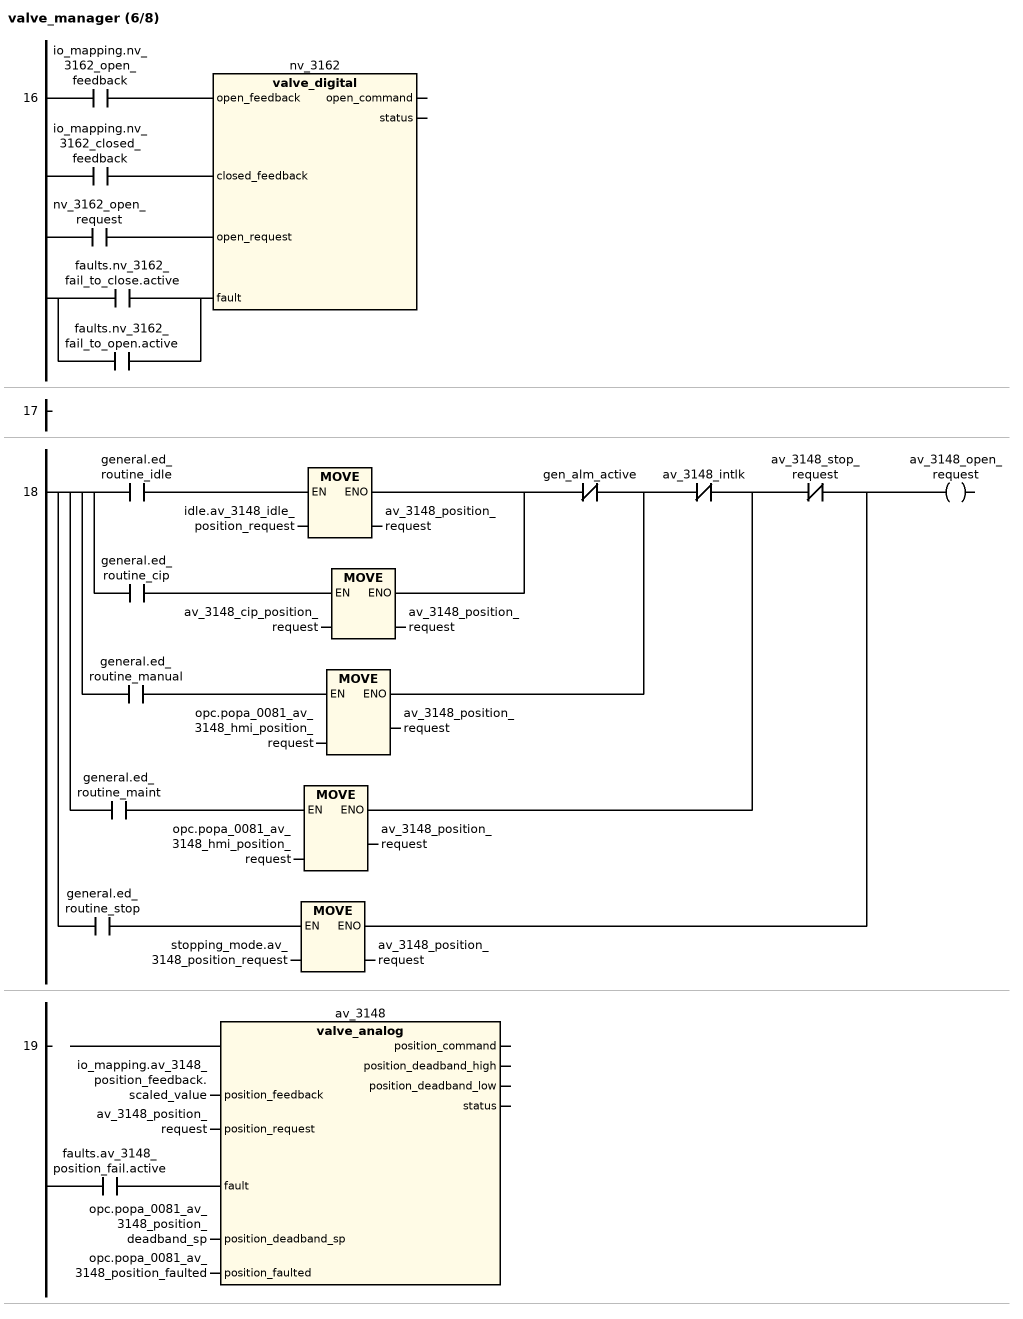
// NETWORK 16
nv_3162(
    open_feedback := io_mapping.nv_3162_open_feedback,
    closed_feedback := io_mapping.nv_3162_closed_feedback,
    open_request := nv_3162_open_request,
    fault := faults.nv_3162_fail_to_close.active OR faults.nv_3162_fail_to_open.active); // valve_digital

// NETWORK 17

// NETWORK 18
_w1 := general.ed_routine_idle;
IF _w1 THEN av_3148_position_request := idle.av_3148_idle_position_request; END_IF
_w2 := general.ed_routine_cip;
IF _w2 THEN av_3148_position_request := av_3148_cip_position_request; END_IF
_w3 := general.ed_routine_manual;
IF _w3 THEN av_3148_position_request := opc.popa_0081_av_3148_hmi_position_request; END_IF
_w4 := general.ed_routine_maint;
IF _w4 THEN av_3148_position_request := opc.popa_0081_av_3148_hmi_position_request; END_IF
_w5 := general.ed_routine_stop;
IF _w5 THEN av_3148_position_request := stopping_mode.av_3148_position_request; END_IF
av_3148_open_request := (((_w1 OR _w2) AND NOT gen_alm_active OR _w3) AND NOT av_3148_intlk OR _w4) AND NOT av_3148_stop_request OR _w5;

// NETWORK 19
av_3148(
    position_feedback := io_mapping.av_3148_position_feedback.scaled_value,
    position_request := av_3148_position_request,
    fault := faults.av_3148_position_fail.active,
    position_deadband_sp := opc.popa_0081_av_3148_position_deadband_sp,
    position_faulted := opc.popa_0081_av_3148_position_faulted); // valve_analog

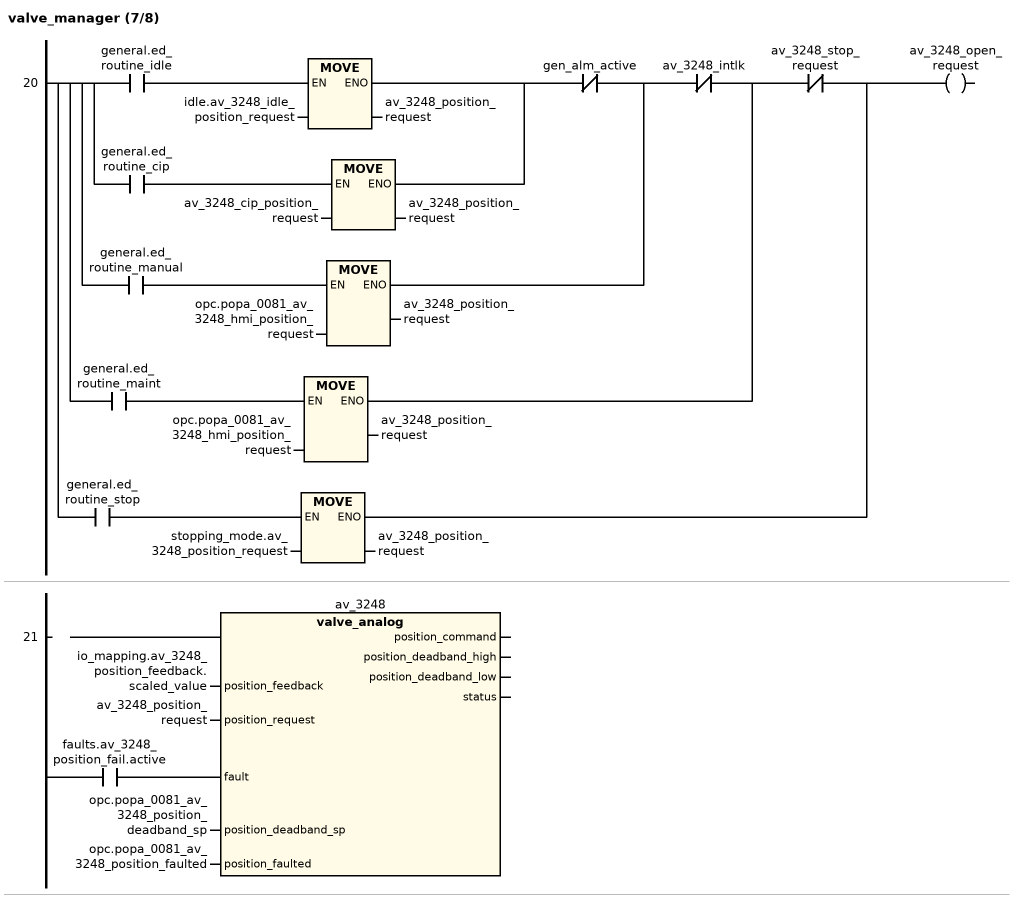
// NETWORK 20
_w6 := general.ed_routine_idle;
IF _w6 THEN av_3248_position_request := idle.av_3248_idle_position_request; END_IF
_w7 := general.ed_routine_cip;
IF _w7 THEN av_3248_position_request := av_3248_cip_position_request; END_IF
_w8 := general.ed_routine_manual;
IF _w8 THEN av_3248_position_request := opc.popa_0081_av_3248_hmi_position_request; END_IF
_w9 := general.ed_routine_maint;
IF _w9 THEN av_3248_position_request := opc.popa_0081_av_3248_hmi_position_request; END_IF
_w10 := general.ed_routine_stop;
IF _w10 THEN av_3248_position_request := stopping_mode.av_3248_position_request; END_IF
av_3248_open_request := (((_w6 OR _w7) AND NOT gen_alm_active OR _w8) AND NOT av_3248_intlk OR _w9) AND NOT av_3248_stop_request OR _w10;

// NETWORK 21
av_3248(
    position_feedback := io_mapping.av_3248_position_feedback.scaled_value,
    position_request := av_3248_position_request,
    fault := faults.av_3248_position_fail.active,
    position_deadband_sp := opc.popa_0081_av_3248_position_deadband_sp,
    position_faulted := opc.popa_0081_av_3248_position_faulted); // valve_analog

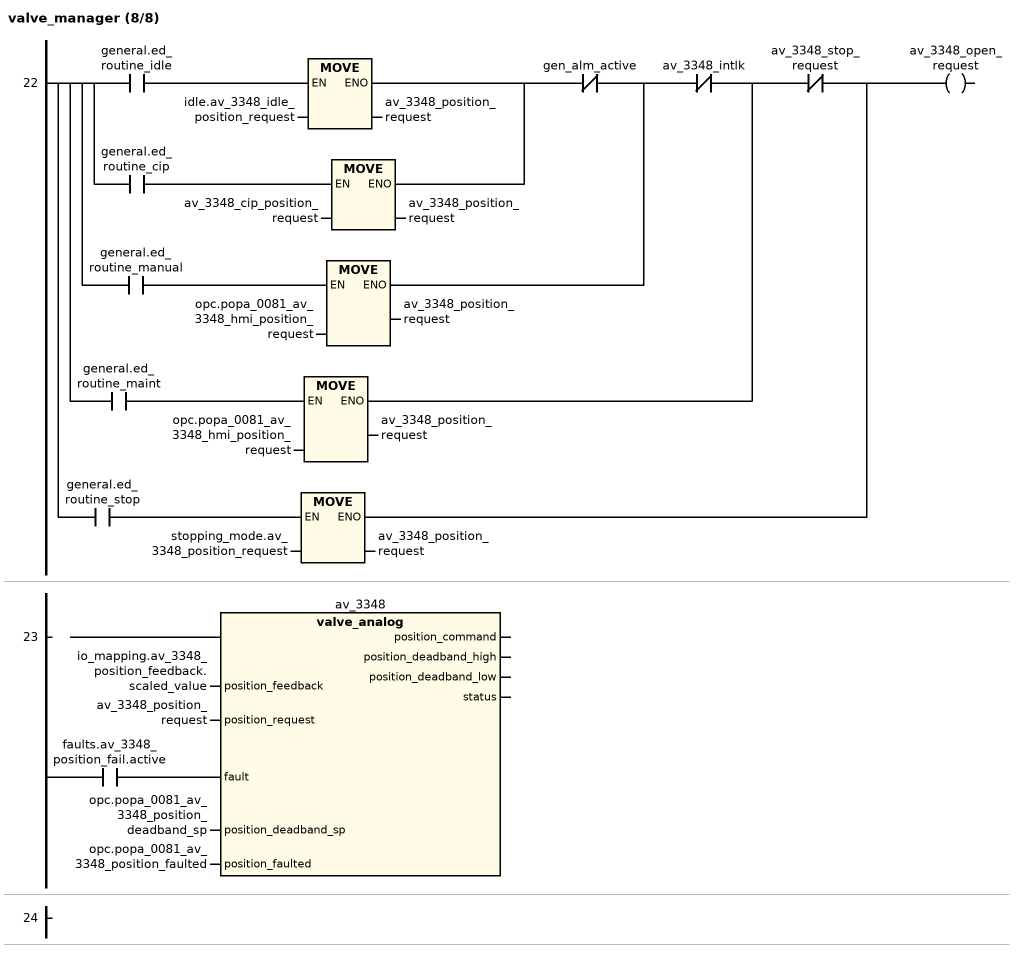
// NETWORK 22
_w11 := general.ed_routine_idle;
IF _w11 THEN av_3348_position_request := idle.av_3348_idle_position_request; END_IF
_w12 := general.ed_routine_cip;
IF _w12 THEN av_3348_position_request := av_3348_cip_position_request; END_IF
_w13 := general.ed_routine_manual;
IF _w13 THEN av_3348_position_request := opc.popa_0081_av_3348_hmi_position_request; END_IF
_w14 := general.ed_routine_maint;
IF _w14 THEN av_3348_position_request := opc.popa_0081_av_3348_hmi_position_request; END_IF
_w15 := general.ed_routine_stop;
IF _w15 THEN av_3348_position_request := stopping_mode.av_3348_position_request; END_IF
av_3348_open_request := (((_w11 OR _w12) AND NOT gen_alm_active OR _w13) AND NOT av_3348_intlk OR _w14) AND NOT av_3348_stop_request OR _w15;

// NETWORK 23
av_3348(
    position_feedback := io_mapping.av_3348_position_feedback.scaled_value,
    position_request := av_3348_position_request,
    fault := faults.av_3348_position_fail.active,
    position_deadband_sp := opc.popa_0081_av_3348_position_deadband_sp,
    position_faulted := opc.popa_0081_av_3348_position_faulted); // valve_analog

// NETWORK 24

END_PROGRAM

// ---- POUs/opc_mapping.TcPOU
PROGRAM opc_mapping
VAR
END_VAR

//This program maps values from the local variable to the OPC readable tag.
//Setpoints should NOT be mapped here.  The OPC tag should be used directly where needed
opc.popa_0081_av_3148_position_fail_active :=faults.av_3148_position_fail.active;
opc.popa_0081_u_3112_fail_to_start_active:=faults.u_3112_fail_to_start.active;
opc.popa_0081_u_3112_fail_to_stop_active:=faults.u_3112_fail_to_stop.active;
opc.popa_0081_u_3160_fail_to_start_active:=faults.u_3160_fail_to_start.active;
opc.popa_0081_u_3160_fail_to_stop_active:=faults.u_3112_fail_to_stop.active;
opc.popa_0081_cpt_3144_low_low_active:=faults.cpt_3144_low_low.active;
opc.popa_0081_cpt_3144_low_active:=faults.cpt_3144_low.active;
opc.popa_0081_cpt_3144_high_active:=faults.cpt_3144_high.active;
opc.popa_0081_cpt_3144_high_high_active:=faults.cpt_3144_high_high.active;

opc.popa_0081_ed_routine_critical_stop := general.ed_critical_stop;
opc.popa_0081_ed_routine_stop := general.ed_routine_stop;
opc.popa_0081_ed_routine_idle := general.ed_routine_idle;
opc.popa_0081_ed_routine_maint := general.ed_routine_maint;
opc.popa_0081_ed_routine_cip := general.ed_routine_cip;

opc.popa_0081_system_date_time_year:=general.system_date_time.year;
opc.popa_0081_system_date_time_month:=general.system_date_time.month;
opc.popa_0081_system_date_time_day:=general.system_date_time.day;
opc.popa_0081_system_date_time_hour:=general.system_date_time.hour;
opc.popa_0081_system_date_time_minute:=general.system_date_time.minute;
opc.popa_0081_system_date_time_second:=general.system_date_time.second;

//---Field Instrumentation---------------------------------------------------------------------------------------------------------------------------
opc.popa_0081_cpt_3144_scaled_value:=io_mapping.cpt_3144.scaled_value;

opc.popa_0081_ft_3122_scaled_value:=io_mapping.ft_3122.scaled_value;
opc.popa_0081_ft_3222_scaled_value:=io_mapping.ft_3222.scaled_value;
opc.popa_0081_ft_3322_scaled_value:=io_mapping.ft_3322.scaled_value;

opc.popa_0081_lt_3102_scaled_value:=io_mapping.lt_3102.scaled_value;
opc.popa_0081_lt_3202_scaled_value:=io_mapping.lt_3202.scaled_value;
opc.popa_0081_lt_3302_scaled_value:=io_mapping.lt_3302.scaled_value;
opc.popa_0081_lt_3153_scaled_value:=io_mapping.lt_3153.scaled_value;
opc.popa_0081_lt_3253_scaled_value:=io_mapping.lt_3253.scaled_value;
opc.popa_0081_lt_3353_scaled_value:=io_mapping.lt_3353.scaled_value;
opc.popa_0091_lt_3402_scaled_value:=io_mapping.lt_3402.scaled_value;

opc.popa_0081_pt_3119_scaled_value:=io_mapping.pt_3119.scaled_value;
opc.popa_0081_pt_3219_scaled_value:=io_mapping.pt_3219.scaled_value;
opc.popa_0081_pt_3319_scaled_value:=io_mapping.pt_3319.scaled_value;
opc.popa_0081_pt_3141_scaled_value:=io_mapping.pt_3141.scaled_value;
opc.popa_0081_pt_3241_scaled_value:=io_mapping.pt_3241.scaled_value;
opc.popa_0081_pt_3341_scaled_value:=io_mapping.pt_3341.scaled_value;
opc.popa_0091_pt_3428_scaled_value:=io_mapping.pt_3428.scaled_value;
opc.popa_0091_pt_3414_scaled_value:=io_mapping.pt_3414.scaled_value;

opc.popa_0081_tt_3118_scaled_value:=io_mapping.tt_3118.scaled_value;
opc.popa_0081_tt_3218_scaled_value:=io_mapping.tt_3218.scaled_value;
opc.popa_0081_tt_3318_scaled_value:=io_mapping.tt_3318.scaled_value;
opc.popa_0081_tt_3140_scaled_value:=io_mapping.tt_3140.scaled_value;
opc.popa_0081_tt_3240_scaled_value:=io_mapping.tt_3240.scaled_value;
opc.popa_0081_tt_3340_scaled_value:=io_mapping.tt_3340.scaled_value;
opc.popa_0091_tt_3432_scaled_value:=io_mapping.tt_3432.scaled_value;

//---Pumps---------------------------------------------------------------------------------------------------------------
opc.popa_0081_u_3112_speed_command_scaled_value:=output_mapping.u_3112_speed_command.scaled_value;
opc.popa_0081_u_3112_speed_feedback_scaled_value:=io_mapping.u_3112_speed_feedback.scaled_value;
opc.popa_0081_u_3112_run_request:=pump_manager.u_3112.run_request;
opc.popa_0081_u_3112_speed_request:=pump_manager.u_3112.speed_request;
opc.popa_0081_u_3112_runtime_today:=pump_manager.u_3112.runtime_today;
opc.popa_0081_u_3112_runtime_total:=pump_manager.u_3112.runtime_total;
opc.popa_0081_u_3112_runtime_maint:=pump_manager.u_3112.runtime_maint;
opc.popa_0081_u_3112_status:=pump_manager.u_3112.status;

opc.popa_0081_u_3212_speed_command_scaled_value:=output_mapping.u_3212_speed_command.scaled_value;
opc.popa_0081_u_3212_speed_feedback_scaled_value:=io_mapping.u_3212_speed_feedback.scaled_value;
opc.popa_0081_u_3212_run_request:=pump_manager.u_3212.run_request;
opc.popa_0081_u_3212_speed_request:=pump_manager.u_3212.speed_request;
opc.popa_0081_u_3212_runtime_today:=pump_manager.u_3212.runtime_today;
opc.popa_0081_u_3212_runtime_total:=pump_manager.u_3212.runtime_total;
opc.popa_0081_u_3212_runtime_maint:=pump_manager.u_3212.runtime_maint;
opc.popa_0081_u_3212_status:=pump_manager.u_3212.status;

opc.popa_0081_u_3312_speed_command_scaled_value:=output_mapping.u_3312_speed_command.scaled_value;
opc.popa_0081_u_3312_speed_feedback_scaled_value:=io_mapping.u_3312_speed_feedback.scaled_value;
opc.popa_0081_u_3312_run_request:=pump_manager.u_3312.run_request;
opc.popa_0081_u_3312_speed_request:=pump_manager.u_3312.speed_request;
opc.popa_0081_u_3312_runtime_today:=pump_manager.u_3312.runtime_today;
opc.popa_0081_u_3312_runtime_total:=pump_manager.u_3312.runtime_total;
opc.popa_0081_u_3312_runtime_maint:=pump_manager.u_3312.runtime_maint;
opc.popa_0081_u_3312_status:=pump_manager.u_3312.status;

opc.popa_0081_u_3160_speed_command_scaled_value:=output_mapping.u_3160_speed_command.scaled_value;
opc.popa_0081_u_3160_speed_feedback_scaled_value:=io_mapping.u_3160_speed_feedback.scaled_value;
opc.popa_0081_u_3160_run_request:=pump_manager.u_3160.run_request;
opc.popa_0081_u_3160_speed_request:=pump_manager.u_3160.speed_request;
opc.popa_0081_u_3160_runtime_today:=pump_manager.u_3160.runtime_today;
opc.popa_0081_u_3160_runtime_total:=pump_manager.u_3160.runtime_total;
opc.popa_0081_u_3160_runtime_maint:=pump_manager.u_3160.runtime_maint;
opc.popa_0081_u_3160_status:=pump_manager.u_3160.status;

opc.popa_0081_u_3260_speed_command_scaled_value:=output_mapping.u_3260_speed_command.scaled_value;
opc.popa_0081_u_3260_speed_feedback_scaled_value:=io_mapping.u_3260_speed_feedback.scaled_value;
opc.popa_0081_u_3260_run_request:=pump_manager.u_3260.run_request;
opc.popa_0081_u_3260_speed_request:=pump_manager.u_3260.speed_request;
opc.popa_0081_u_3260_runtime_today:=pump_manager.u_3260.runtime_today;
opc.popa_0081_u_3260_runtime_total:=pump_manager.u_3260.runtime_total;
opc.popa_0081_u_3260_runtime_maint:=pump_manager.u_3260.runtime_maint;
opc.popa_0081_u_3260_status:=pump_manager.u_3260.status;

opc.popa_0081_u_3360_speed_command_scaled_value:=output_mapping.u_3360_speed_command.scaled_value;
opc.popa_0081_u_3360_speed_feedback_scaled_value:=io_mapping.u_3360_speed_feedback.scaled_value;
opc.popa_0081_u_3360_run_request:=pump_manager.u_3360.run_request;
opc.popa_0081_u_3360_speed_request:=pump_manager.u_3360.speed_request;
opc.popa_0081_u_3360_runtime_today:=pump_manager.u_3360.runtime_today;
opc.popa_0081_u_3360_runtime_total:=pump_manager.u_3360.runtime_total;
opc.popa_0081_u_3360_runtime_maint:=pump_manager.u_3360.runtime_maint;
opc.popa_0081_u_3360_status:=pump_manager.u_3360.status;

opc.popa_0081_u_3370_speed_command_scaled_value:=output_mapping.u_3370_speed_command.scaled_value;
opc.popa_0081_u_3370_speed_feedback_scaled_value:=io_mapping.u_3370_speed_feedback.scaled_value;
opc.popa_0081_u_3370_run_request:=pump_manager.u_3370.run_request;
opc.popa_0081_u_3370_speed_request:=pump_manager.u_3370.speed_request;
opc.popa_0081_u_3370_runtime_today:=pump_manager.u_3370.runtime_today;
opc.popa_0081_u_3370_runtime_total:=pump_manager.u_3370.runtime_total;
opc.popa_0081_u_3370_runtime_maint:=pump_manager.u_3370.runtime_maint;
opc.popa_0081_u_3370_status:=pump_manager.u_3370.status;

opc.popa_0091_u_3405_speed_command_scaled_value:=output_mapping.u_3405_speed_command.scaled_value;
opc.popa_0091_u_3405_speed_feedback_scaled_value:=io_mapping.u_3405_speed_feedback.scaled_value;
opc.popa_0091_u_3405_run_request:=pump_manager.u_3405.run_request;
opc.popa_0091_u_3405_speed_request:=pump_manager.u_3405.speed_request;
opc.popa_0091_u_3405_runtime_today:=pump_manager.u_3405.runtime_today;
opc.popa_0091_u_3405_runtime_total:=pump_manager.u_3405.runtime_total;
opc.popa_0091_u_3405_runtime_maint:=pump_manager.u_3405.runtime_maint;
opc.popa_0091_u_3405_status:=pump_manager.u_3405.status;



//---Valves------------------------------------------------------------------------------------------------------------------

opc.popa_0081_av_3148_position_feedback_scaled_value:=io_mapping.av_3148_position_feedback.scaled_value;
opc.popa_0081_av_3148_position_command_scaled_value:=output_mapping.av_3148_position_command.scaled_value;
opc.popa_0081_av_3148_position_feedback:=valve_manager.av_3148.position_feedback;
opc.popa_0081_av_3148_position_request:=valve_manager.av_3148.position_request;
opc.popa_0081_av_3148_status:=valve_manager.av_3148.status;

opc.popa_0081_av_3248_position_feedback_scaled_value:=io_mapping.av_3248_position_feedback.scaled_value;
opc.popa_0081_av_3248_position_command_scaled_value:=output_mapping.av_3248_position_command.scaled_value;
opc.popa_0081_av_3248_position_feedback:=valve_manager.av_3248.position_feedback;
opc.popa_0081_av_3248_position_request:=valve_manager.av_3248.position_request;
opc.popa_0081_av_3248_status:=valve_manager.av_3248.status;

opc.popa_0081_av_3348_position_feedback_scaled_value:=io_mapping.av_3348_position_feedback.scaled_value;
opc.popa_0081_av_3348_position_command_scaled_value:=output_mapping.av_3348_position_command.scaled_value;
opc.popa_0081_av_3348_position_feedback:=valve_manager.av_3348.position_feedback;
opc.popa_0081_av_3348_position_request:=valve_manager.av_3348.position_request;
opc.popa_0081_av_3348_status:=valve_manager.av_3348.status;
(*
opc.popa_0081_u_3160_run_request:=motor_starter_control.u_3160.run_request;
opc.popa_0081_u_3160_runtime_today:=motor_starter_control.u_3160.runtime_today;
opc.popa_0081_u_3160_runtime_total:=motor_starter_control.u_3160.runtime_total;
opc.popa_0081_u_3160_runtime_maint:=motor_starter_control.u_3160.runtime_maint;
opc.popa_0081_u_3160_status:=motor_starter_control.u_3160.status;
*)


opc.popa_0081_nv_3110_open_request:=valve_manager.nv_3110.open_request;
opc.popa_0081_nv_3110_status:=valve_manager.nv_3110.status;
opc.popa_0081_nv_3110_fail_to_open_active :=faults.nv_3110_fail_to_open.active;
opc.popa_0081_nv_3110_fail_to_close_active :=faults.nv_3110_fail_to_close.active;

opc.popa_0081_nv_3210_open_request:=valve_manager.nv_3210.open_request;
opc.popa_0081_nv_3210_status:=valve_manager.nv_3210.status;
opc.popa_0081_nv_3210_fail_to_open_active :=faults.nv_3210_fail_to_open.active;
opc.popa_0081_nv_3210_fail_to_close_active :=faults.nv_3210_fail_to_close.active;

opc.popa_0081_nv_3310_open_request:=valve_manager.nv_3310.open_request;
opc.popa_0081_nv_3310_status:=valve_manager.nv_3310.status;
opc.popa_0081_nv_3310_fail_to_open_active :=faults.nv_3310_fail_to_open.active;
opc.popa_0081_nv_3310_fail_to_close_active :=faults.nv_3310_fail_to_close.active;

opc.popa_0081_nv_3135_open_request:=valve_manager.nv_3135.open_request;
opc.popa_0081_nv_3135_status:=valve_manager.nv_3135.status;
opc.popa_0081_nv_3135_fail_to_open_active :=faults.nv_3135_fail_to_open.active;
opc.popa_0081_nv_3135_fail_to_close_active :=faults.nv_3135_fail_to_close.active;

opc.popa_0081_nv_3235_open_request:=valve_manager.nv_3235.open_request;
opc.popa_0081_nv_3235_status:=valve_manager.nv_3235.status;
opc.popa_0081_nv_3235_fail_to_open_active :=faults.nv_3235_fail_to_open.active;
opc.popa_0081_nv_3235_fail_to_close_active :=faults.nv_3235_fail_to_close.active;

opc.popa_0081_nv_3335_open_request:=valve_manager.nv_3335.open_request;
opc.popa_0081_nv_3335_status:=valve_manager.nv_3335.status;
opc.popa_0081_nv_3335_fail_to_open_active :=faults.nv_3335_fail_to_open.active;
opc.popa_0081_nv_3335_fail_to_close_active :=faults.nv_3335_fail_to_close.active;

opc.popa_0081_nv_3372_open_request:=valve_manager.nv_3372.open_request;
opc.popa_0081_nv_3372_status:=valve_manager.nv_3372.status;
opc.popa_0081_nv_3372_fail_to_open_active :=faults.nv_3372_fail_to_open.active;
opc.popa_0081_nv_3372_fail_to_close_active :=faults.nv_3372_fail_to_close.active;

//opc.popa_0081_nv_3162_hmi_open_request:=valve_manager.nv_3162.open_request;
opc.popa_0081_nv_3162_open_request:=valve_manager.nv_3162.open_request;
opc.popa_0081_nv_3162_status:=valve_manager.nv_3162.status;
opc.popa_0081_nv_3162_fail_to_open_active :=faults.nv_3162_fail_to_open.active;
opc.popa_0081_nv_3162_fail_to_close_active :=faults.nv_3162_fail_to_close.active;

END_PROGRAM

// ---- POUs/output_mapping.TcPOU
PROGRAM output_mapping
VAR PERSISTENT
	//Motor vfd speed command function block
	u_3112_speed_command : analog_scaling;
	u_3212_speed_command : analog_scaling;
	u_3312_speed_command : analog_scaling;
	u_3160_speed_command : analog_scaling;
	u_3260_speed_command : analog_scaling;
	u_3360_speed_command : analog_scaling;
	u_3370_speed_command : analog_scaling;
	u_3405_speed_command : analog_scaling;
	
	//Analog valve position command
	av_3148_position_command : analog_scaling;
	av_3248_position_command : analog_scaling;
	av_3348_position_command : analog_scaling;
	nv_3110_position_command : analog_scaling;
	nv_3210_position_command : analog_scaling;
	nv_3310_position_command : analog_scaling;
	//Motor vfd speed command scaled output, mappped to a physical output
	{attribute 'TcLinkTo' := 'TIID^Device 1 (EtherCAT)^Term 1 (EK1200)^Term 4 (EL4124)^AO Output Channel 1^Analog output'}
	u_3112_speed_command_io AT %Q* : INT;
	{attribute 'TcLinkTo' := 'TIID^Device 1 (EtherCAT)^Term 1 (EK1200)^Term 4 (EL4124)^AO Output Channel 2^Analog output'}
	u_3212_speed_command_io AT %Q* : INT;
	{attribute 'TcLinkTo' := 'TIID^Device 1 (EtherCAT)^Term 1 (EK1200)^Term 4 (EL4124)^AO Output Channel 3^Analog output'}
	u_3312_speed_command_io AT %Q* : INT;
	{attribute 'TcLinkTo' := 'TIID^Device 1 (EtherCAT)^Term 1 (EK1200)^Term 4 (EL4124)^AO Output Channel 4^Analog output'}
	u_3160_speed_command_io AT %Q* : INT;
	{attribute 'TcLinkTo' := 'TIID^Device 1 (EtherCAT)^Term 1 (EK1200)^Term 5 (EL4124)^AO Output Channel 1^Analog output'}
	u_3260_speed_command_io AT %Q* : INT;
	{attribute 'TcLinkTo' := 'TIID^Device 1 (EtherCAT)^Term 1 (EK1200)^Term 5 (EL4124)^AO Output Channel 2^Analog output'}
	u_3360_speed_command_io AT %Q* : INT;
	{attribute 'TcLinkTo' := 'TIID^Device 1 (EtherCAT)^Term 1 (EK1200)^Term 5 (EL4124)^AO Output Channel 3^Analog output'}
	u_3370_speed_command_io AT %Q* : INT;
	{attribute 'TcLinkTo' := 'TIID^Device 1 (EtherCAT)^Term 40 (EK1100)^Term 42 (EL4124)^AO Output Channel 1^Analog output'}
	u_3405_speed_command_io AT %Q* : INT;
	
	//Motor vfd run command, mapped to a physical output
	{attribute 'TcLinkTo' :=  'TIID^Device 1 (EtherCAT)^Term 1 (EK1200)^Term 7 (EL1859)^Channel 9^Output'}
	u_3112_run_command_io AT %Q* : BOOL;
	{attribute 'TcLinkTo' :=  'TIID^Device 1 (EtherCAT)^Term 1 (EK1200)^Term 7 (EL1859)^Channel 11^Output'}
	u_3212_run_command_io AT %Q* : BOOL;
	{attribute 'TcLinkTo' :=  'TIID^Device 1 (EtherCAT)^Term 1 (EK1200)^Term 7 (EL1859)^Channel 13^Output'}
	u_3312_run_command_io AT %Q* : BOOL;
	{attribute 'TcLinkTo' :=  'TIID^Device 1 (EtherCAT)^Term 1 (EK1200)^Term 7 (EL1859)^Channel 15^Output'}	
	u_3160_run_command_io AT %Q* : BOOL;
	{attribute 'TcLinkTo' :=  'TIID^Device 1 (EtherCAT)^Term 1 (EK1200)^Term 8 (EL1859)^Channel 9^Output'}
	u_3260_run_command_io AT %Q* : BOOL;
	{attribute 'TcLinkTo' :=  'TIID^Device 1 (EtherCAT)^Term 1 (EK1200)^Term 8 (EL1859)^Channel 11^Output'}
	u_3360_run_command_io AT %Q* : BOOL;
	{attribute 'TcLinkTo' :=  'TIID^Device 1 (EtherCAT)^Term 1 (EK1200)^Term 8 (EL1859)^Channel 13^Output'}
	u_3370_run_command_io AT %Q* : BOOL;
	{attribute 'TcLinkTo' :=  'TIID^Device 1 (EtherCAT)^Term 40 (EK1100)^Term 43 (EL1859)^Channel 9^Output'}
	u_3405_run_command_io AT %Q* : BOOL;
	
	//Motor Fault Reset
	{attribute 'TcLinkTo' :=  'TIID^Device 1 (EtherCAT)^Term 1 (EK1200)^Term 7 (EL1859)^Channel 10^Output'}
	u_3112_fault_reset_io AT %Q* : BOOL;
	{attribute 'TcLinkTo' :=  'TIID^Device 1 (EtherCAT)^Term 1 (EK1200)^Term 7 (EL1859)^Channel 12^Output'}
	u_3212_fault_reset_io AT %Q* : BOOL;
	{attribute 'TcLinkTo' :=  'TIID^Device 1 (EtherCAT)^Term 1 (EK1200)^Term 7 (EL1859)^Channel 14^Output'}
	u_3312_fault_reset_io AT %Q* : BOOL;
	{attribute 'TcLinkTo' :=  'TIID^Device 1 (EtherCAT)^Term 1 (EK1200)^Term 7 (EL1859)^Channel 16^Output'}
	u_3160_fault_reset_io AT %Q* : BOOL;
	{attribute 'TcLinkTo' :=  'TIID^Device 1 (EtherCAT)^Term 1 (EK1200)^Term 8 (EL1859)^Channel 10^Output'}
	u_3260_fault_reset_io AT %Q* : BOOL;
	{attribute 'TcLinkTo' :=  'TIID^Device 1 (EtherCAT)^Term 1 (EK1200)^Term 8 (EL1859)^Channel 12^Output'}
	u_3360_fault_reset_io AT %Q* : BOOL;
	{attribute 'TcLinkTo' :=  'TIID^Device 1 (EtherCAT)^Term 1 (EK1200)^Term 8 (EL1859)^Channel 14^Output'}
	u_3370_fault_reset_io AT %Q* : BOOL;
	{attribute 'TcLinkTo' :=  'TIID^Device 1 (EtherCAT)^Term 40 (EK1100)^Term 43 (EL1859)^Channel 10^Output'}
	u_3405_fault_reset_io AT %Q* : BOOL;
	
		
	//Analog valve position command output valve
	{attribute 'TcLinkTo' := 'TIID^Device 1 (EtherCAT)^Term 20 (EK1100-0018)^Term 26 (EL4124)^AO Output Channel 1^Analog output'}
	av_3148_position_command_io AT %Q* : INT;
	{attribute 'TcLinkTo' := 'TIID^Device 1 (EtherCAT)^Term 20 (EK1100-0018)^Term 26 (EL4124)^AO Output Channel 2^Analog output'}
	av_3248_position_command_io AT %Q* : INT;
	{attribute 'TcLinkTo' := 'TIID^Device 1 (EtherCAT)^Term 20 (EK1100-0018)^Term 26 (EL4124)^AO Output Channel 3^Analog output'}
	av_3348_position_command_io AT %Q* : INT;
	
		//Digital valve open command
	{attribute 'TcLinkTo' := 'TIID^Device 1 (EtherCAT)^Term 31 (EK1914)^Term 32 (EL1859)^Channel 11^Output'}
	nv_3110_open_command_io AT %Q* : BOOL;
	{attribute 'TcLinkTo' := 'TIID^Device 1 (EtherCAT)^Term 31 (EK1914)^Term 32 (EL1859)^Channel 10^Output'}
	nv_3210_open_command_io AT %Q* : BOOL;
	{attribute 'TcLinkTo' := 'TIID^Device 1 (EtherCAT)^Term 31 (EK1914)^Term 32 (EL1859)^Channel 13^Output'}
	nv_3310_open_command_io AT %Q* : BOOL;
	{attribute 'TcLinkTo' := 'TIID^Device 1 (EtherCAT)^Term 31 (EK1914)^Term 32 (EL1859)^Channel 12^Output'}
	nv_3135_open_command_io AT %Q* : BOOL;
	{attribute 'TcLinkTo' := 'TIID^Device 1 (EtherCAT)^Term 31 (EK1914)^Term 32 (EL1859)^Channel 14^Output'}
	nv_3235_open_command_io AT %Q* : BOOL;
	{attribute 'TcLinkTo' := 'TIID^Device 1 (EtherCAT)^Term 31 (EK1914)^Term 32 (EL1859)^Channel 15^Output'}
	nv_3335_open_command_io AT %Q* : BOOL;
	{attribute 'TcLinkTo' := 'TIID^Device 1 (EtherCAT)^Term 31 (EK1914)^Term 32 (EL1859)^Channel 16^Output'}
	nv_3372_open_command_io AT %Q* : BOOL;
	{attribute 'TcLinkTo' := 'TIID^Device 1 (EtherCAT)^Term 31 (EK1914)^Term 32 (EL1859)^Channel 9^Output'}
	nv_3162_open_command_io AT %Q* : BOOL;
	
	safety_reset AT %Q* : BOOL;
END_VAR

//Map the motor run command to the command output
u_3112_run_command_io:=pump_manager.u_3112.run_command;
u_3212_run_command_io:=pump_manager.u_3212.run_command;
u_3312_run_command_io:=pump_manager.u_3312.run_command;
u_3160_run_command_io:=pump_manager.u_3160.run_command;
u_3260_run_command_io:=pump_manager.u_3260.run_command;
u_3360_run_command_io:=pump_manager.u_3360.run_command;
u_3370_run_command_io:=pump_manager.u_3370.run_command;
u_3405_run_command_io:=pump_manager.u_3405.run_command;

//Instantiate u_3112 Speed command analog output function block
u_3112_speed_command();
//Map values from the OPC GVL so that they can be written to from outside POU(IE from HMI)
u_3112_speed_command.eu_max:=32767;
u_3112_speed_command.eu_min:=0;
u_3112_speed_command.filter_factor:=opc.popa_0081_u_3112_speed_command_filter_factor;
u_3112_speed_command.raw_max:=60;
u_3112_speed_command.raw_min:=0;

//Map output from motor control pou to scaling block
u_3112_speed_command.raw_input := pump_manager.u_3112.speed_command;

//Map the analog scaling function block raw input to the physical raw output variable
u_3112_speed_command_io := REAL_TO_INT(u_3112_speed_command.scaled_value);

//Instantiate Example analog output function block
u_3212_speed_command();
//Map values from the OPC GVL so that they can be written to from outside POU(IE from HMI)
u_3212_speed_command.eu_max:=32767;
u_3212_speed_command.eu_min:=0;
u_3212_speed_command.filter_factor:=opc.popa_0081_u_3212_speed_command_filter_factor;
u_3212_speed_command.raw_max:=60;
u_3212_speed_command.raw_min:=0;

//Map output from motor control pou to scaling block
u_3212_speed_command.raw_input := pump_manager.u_3212.speed_command;

//Map the analog scaling function block raw input to the physical raw output variable
u_3212_speed_command_io := REAL_TO_INT(u_3212_speed_command.scaled_value);


//Instantiate Example analog output function block
u_3312_speed_command();
//Map values from the OPC GVL so that they can be written to from outside POU(IE from HMI)
u_3312_speed_command.eu_max:=32767;
u_3312_speed_command.eu_min:=0;
u_3312_speed_command.filter_factor:=opc.popa_0081_u_3312_speed_command_filter_factor;
u_3312_speed_command.raw_max:=60;
u_3312_speed_command.raw_min:=0;

//Map output from motor control pou to scaling block
u_3312_speed_command.raw_input := pump_manager.u_3312.speed_command;

//Map the analog scaling function block raw input to the physical raw output variable
u_3312_speed_command_io := REAL_TO_INT(u_3312_speed_command.scaled_value);


//Instantiate Example analog output function block
u_3160_speed_command();
//Map values from the OPC GVL so that they can be written to from outside POU(IE from HMI)
u_3160_speed_command.eu_max:=32767;
u_3160_speed_command.eu_min:=0;
u_3160_speed_command.filter_factor:=opc.popa_0081_u_3160_speed_command_filter_factor;
u_3160_speed_command.raw_max:=60;
u_3160_speed_command.raw_min:=0;

//Map output from motor control pou to scaling block
u_3160_speed_command.raw_input := pump_manager.u_3160.speed_command;

//Map the analog scaling function block raw input to the physical raw output variable
u_3160_speed_command_io := REAL_TO_INT(u_3160_speed_command.scaled_value);

//Instantiate Example analog output function block
u_3260_speed_command();
//Map values from the OPC GVL so that they can be written to from outside POU(IE from HMI)
u_3260_speed_command.eu_max:=32767;
u_3260_speed_command.eu_min:=0;
u_3260_speed_command.filter_factor:=opc.popa_0081_u_3260_speed_command_filter_factor;
u_3260_speed_command.raw_max:=60;
u_3260_speed_command.raw_min:=0;

//Map output from motor control pou to scaling block
u_3260_speed_command.raw_input := pump_manager.u_3260.speed_command;

//Map the analog scaling function block raw input to the physical raw output variable
u_3260_speed_command_io := REAL_TO_INT(u_3260_speed_command.scaled_value);

//Instantiate Example analog output function block
u_3360_speed_command();
//Map values from the OPC GVL so that they can be written to from outside POU(IE from HMI)
u_3360_speed_command.eu_max:=32767;
u_3360_speed_command.eu_min:=0;
u_3360_speed_command.filter_factor:=opc.popa_0081_u_3360_speed_command_filter_factor;
u_3360_speed_command.raw_max:=60;
u_3360_speed_command.raw_min:=0;

//Map output from motor control pou to scaling block
u_3360_speed_command.raw_input := pump_manager.u_3360.speed_command;

//Map the analog scaling function block raw input to the physical raw output variable
u_3360_speed_command_io := REAL_TO_INT(u_3360_speed_command.scaled_value);


//Instantiate Example analog output function block
u_3370_speed_command();
//Map values from the OPC GVL so that they can be written to from outside POU(IE from HMI)
u_3370_speed_command.eu_max:=32767;
u_3370_speed_command.eu_min:=0;
u_3370_speed_command.filter_factor:=opc.popa_0081_u_3370_speed_command_filter_factor;
u_3370_speed_command.raw_max:=60;
u_3370_speed_command.raw_min:=0;

//Map output from motor control pou to scaling block
u_3370_speed_command.raw_input := pump_manager.u_3370.speed_command;

//Map the analog scaling function block raw input to the physical raw output variable
u_3370_speed_command_io := REAL_TO_INT(u_3370_speed_command.scaled_value);

//Instantiate Example analog output function block
u_3405_speed_command();
//Map values from the OPC GVL so that they can be written to from outside POU(IE from HMI)
u_3405_speed_command.eu_max:=32767;
u_3405_speed_command.eu_min:=0;
u_3405_speed_command.filter_factor:=opc.popa_0091_u_3405_speed_command_filter_factor;
u_3405_speed_command.raw_max:=60;
u_3405_speed_command.raw_min:=0;

//Map output from motor control pou to scaling block
u_3405_speed_command.raw_input := pump_manager.u_3405.speed_command;

//Map the analog scaling function block raw input to the physical raw output variable
u_3405_speed_command_io := REAL_TO_INT(u_3405_speed_command.scaled_value);

//Instantiate av_3148 analog output function block
av_3148_position_command();
//Map values from the OPC GVL so that they can be written to from outside POU(IE from HMI)
av_3148_position_command.eu_max:=32767;
av_3148_position_command.eu_min:=0;
av_3148_position_command.filter_factor:=opc.popa_0081_av_3148_position_command_filter_factor;
av_3148_position_command.raw_max:=100;
av_3148_position_command.raw_min:=0;
//Map output from valve control pou to scaling block
av_3148_position_command.raw_input:=valve_manager.av_3148.Position_Command;
//Map the analog scaling function block raw input to the physical raw output variable
av_3148_position_command_io := REAL_TO_INT(av_3148_position_command.scaled_value);

//Instantiate av_3248 analog output function block
av_3248_position_command();
//Map values from the OPC GVL so that they can be written to from outside POU(IE from HMI)
av_3248_position_command.eu_max:=32767;
av_3248_position_command.eu_min:=0;
av_3248_position_command.filter_factor:=opc.popa_0081_av_3248_position_command_filter_factor;
av_3248_position_command.raw_max:=100;
av_3248_position_command.raw_min:=0;
//Map output from valve control pou to scaling block
av_3248_position_command.raw_input:=valve_manager.av_3248.Position_Command;
//Map the analog scaling function block raw input to the physical raw output variable
av_3248_position_command_io := REAL_TO_INT(av_3248_position_command.scaled_value);

//Instantiate av_3348 analog output function block
av_3348_position_command();
//Map values from the OPC GVL so that they can be written to from outside POU(IE from HMI)
av_3348_position_command.eu_max:=32767;
av_3348_position_command.eu_min:=0;
av_3348_position_command.filter_factor:=opc.popa_0081_av_3348_position_command_filter_factor;
av_3348_position_command.raw_max:=100;
av_3348_position_command.raw_min:=0;
//Map output from valve control pou to scaling block
av_3348_position_command.raw_input:=valve_manager.av_3348.Position_Command;
//Map the analog scaling function block raw input to the physical raw output variable
av_3348_position_command_io := REAL_TO_INT(av_3348_position_command.scaled_value);


//Map the digital valve open command to the command output
nv_3110_open_command_io:=valve_manager.nv_3110.open_command;
nv_3210_open_command_io:=valve_manager.nv_3210.open_command;
nv_3310_open_command_io:=valve_manager.nv_3310.open_command;
nv_3135_open_command_io:=valve_manager.nv_3135.open_command;
nv_3235_open_command_io:=valve_manager.nv_3235.open_command;
nv_3335_open_command_io:=valve_manager.nv_3335.open_command;
nv_3372_open_command_io:=valve_manager.nv_3372.open_command;
nv_3162_open_command_io:=valve_manager.nv_3162.open_command;

END_PROGRAM
